// TIA Portal V19 program export: 0 tag tables, 0 data types, 0 data blocks, 3 code blocks (in call order from the OBs), 0 instance data blocks

ORGANIZATION_BLOCK "Main"   // OB1, LAD, ProgramCycle
TITLE = "Main Program Sweep (Cycle)"
{ S7_Optimized_Access := 'TRUE' }
VERSION : 0.1
// stored: AutoNumber true, IsIECCheckEnabled false, SetENOAutomatically false
   VAR_INPUT
      Initial_Call : Bool;   // Initial call of this OB
      Remanence : Bool;   // =True, if remanent data are available
   END_VAR
BEGIN
END_ORGANIZATION_BLOCK

FUNCTION_BLOCK "FB_PumpDown"   // FB3, SCL
{ S7_Optimized_Access := 'TRUE' }
VERSION : 0.1
// Roughing pump-down sequence.
//  generated by LADDER - do not edit by hand
// stored: AutoNumber true, IsIECCheckEnabled false, IsRetainMemResEnabled false, MemoryReserve 100, SetENOAutomatically false, UDAEnableTagReadback false
   VAR
      stable_ok : Bool;   // Pressure stable timer done
      T_stable_t { S7_SetPoint := 'True'} : TON_TIME;   // instance for timer T_stable
   END_VAR
BEGIN
       // timer TON T_stable: Pressure must hold for 10 s before declaring vacuum.
       #T_stable_t(IN := "pressure_ok",
                   PT := T#10s);
       #stable_ok := #T_stable_t.Q;
       // state_machine SM_pumpdown: IDLE -> PUMPING -> AT_VACUUM, with fault fallback.
       CASE "pumpdown_state" OF
           0:  (* IDLE *)
               "pump_start_cmd" := FALSE;
               "at_vacuum" := FALSE;
               IF "pumpdown_request" THEN
                   "pumpdown_state" := 1;
               END_IF;
           1:  (* PUMPING *)
               "pump_start_cmd" := TRUE;
               IF "pump_fault_alarm" THEN
                   "pumpdown_state" := 99;
               ELSIF #stable_ok THEN
                   "pumpdown_state" := 2;
               END_IF;
           2:  (* AT_VACUUM *)
               "at_vacuum" := TRUE;
               IF NOT "pressure_ok" THEN
                   "pumpdown_state" := 1;
               ELSIF NOT "pumpdown_request" THEN
                   "pumpdown_state" := 0;
               END_IF;
           99:  (* FAULT *)
               "pump_start_cmd" := FALSE;
               "at_vacuum" := FALSE;
               IF "reset_pb" AND NOT "pump_fault_alarm" THEN
                   "pumpdown_state" := 0;
               END_IF;
       END_CASE;
END_FUNCTION_BLOCK

FUNCTION_BLOCK "FB_SafetyPermissives"   // FB2, SCL
{ S7_Optimized_Access := 'TRUE' }
VERSION : 0.1
// Interlocks and alarms; runs every scan.
//  generated by LADDER - do not edit by hand
// stored: AutoNumber true, IsIECCheckEnabled false, IsRetainMemResEnabled false, MemoryReserve 100, SetENOAutomatically false, UDAEnableTagReadback false
   VAR
      IL_shutter_rst_mem : Bool;   // edge memory for reset_pb
      ALM_vacuum_ton { S7_SetPoint := 'True'} : TON_TIME;   // on-delay for alarm ALM_vacuum
      ALM_vacuum_ack_mem : Bool;   // edge memory for ack_pb
      ALM_pump_fb_ton { S7_SetPoint := 'True'} : TON_TIME;   // on-delay for alarm ALM_pump_fb
      ALM_pump_fb_ack_mem : Bool;   // edge memory for ack_pb
   END_VAR
BEGIN
       // interlock IL_shutter: Beam shutter permissive - trips on vacuum or valve fault.
       IF NOT ("pressure_ok" AND "gate_valve_closed") THEN
           "beam_shutter_permit" := FALSE;
       END_IF;
       IF "reset_pb" AND NOT #IL_shutter_rst_mem AND ("pressure_ok" AND "gate_valve_closed") THEN
           "beam_shutter_permit" := TRUE;
       END_IF;
       #IL_shutter_rst_mem := "reset_pb";
       // alarm [critical] ALM_vacuum: Vacuum lost (debounced 2 s), latched until acknowledged.
       #ALM_vacuum_ton(IN := NOT "pressure_ok",
                       PT := T#2s);
       IF #ALM_vacuum_ton.Q THEN
           "vacuum_alarm" := TRUE;
       END_IF;
       IF "ack_pb" AND NOT #ALM_vacuum_ack_mem AND NOT #ALM_vacuum_ton.Q THEN
           "vacuum_alarm" := FALSE;
       END_IF;
       #ALM_vacuum_ack_mem := "ack_pb";
       // alarm [alarm] ALM_pump_fb: Pump commanded but no running feedback within 5 s.
       #ALM_pump_fb_ton(IN := "pump_start_cmd" AND NOT "pump_running_fb",
                        PT := T#5s);
       IF #ALM_pump_fb_ton.Q THEN
           "pump_fault_alarm" := TRUE;
       END_IF;
       IF "ack_pb" AND NOT #ALM_pump_fb_ack_mem AND NOT #ALM_pump_fb_ton.Q THEN
           "pump_fault_alarm" := FALSE;
       END_IF;
       #ALM_pump_fb_ack_mem := "ack_pb";
END_FUNCTION_BLOCK
